SUBAPPLICATION Uebung_171c_ASR (* Exercise for ASR_AX_SR, ueber AE-Adapter mit logiBUS_IEA statt logiBUS_IE+AE_EVENT_TO_E *)
  (* Standard: 61499-2; Description: Copyright (c) 2026 Meisterschulen am Ostbahnhof This program and the accompanying materials are made available under the terms of the Eclipse Public License 2.0 which is available at https://www.eclipse.org/legal/epl-2.0/ SPDX-License-Identifier: EPL-2.0 *)
  (* Version 1.0, 2026-09-07, Franz Höpfinger, Meisterschulen am Ostbahnhof, initial API and implementation and/or initial documentation *)
  PACKAGE Uebungen;
  IMPORT logiBUS::io::DI::logiBUS_DI::Input_I1;
  IMPORT logiBUS::io::DI::logiBUS_DI::Input_I2;
  IMPORT logiBUS::io::DI::logiBUS_DI_Events::BUTTON_SINGLE_CLICK;
  IMPORT logiBUS::io::DQ::logiBUS_DO::Output_Q1;
  (* Documentation:
  SET/RESET über AE-Adapter mit logiBUS_IEA (AE bereits eingebaut)
   Dieselbe Funktion wie Uebung_171b_ASR, aber ohne die manuelle AE_EVENT_TO_E-Brücke pro Kanal: logiBUS_IEA ersetzt logiBUS_IE und liefert den AE-Plug (IN) bereits eingebaut - intern verdrahtet logiBUS_IEA genau das, was in 171b noch von Hand mit AE_EVENT_TO_E gebaut wurde.
   Funktionsbeschreibung
    - logiBUS_IEA kapselt intern einen logiBUS_IE und leitet dessen Klick-Events direkt auf einen eigenen AE-Plug (IN) um - derselbe Mechanismus wie IX → IXA für Pegelsignale, nur für Event-Eingänge.
   - ASR_2AE_TO_SR_1 bekommt seine SET_IN/RESET_IN jetzt direkt von den beiden logiBUS_IEA-Instanzen, ohne Zwischenbaustein.
    Arbeitsauftrag
   Testen Sie identisch zu Uebung_171_ASR/Uebung_171b_ASR: I1 klicken → Q1 EIN, I2 klicken → Q1 AUS. Vergleichen Sie alle drei SubApps im Editor: gleiches Verhalten, aber Uebung_171c_ASR kommt mit den wenigsten Bausteinen aus.
  *)
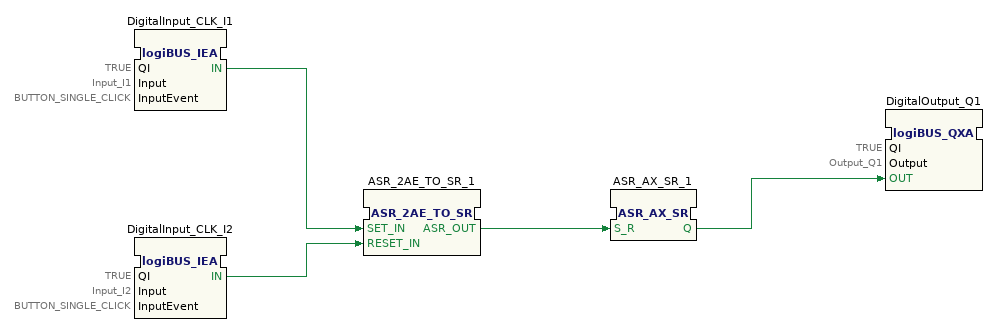
  (* Vergleich zu Uebung_171b_ASR: dort baute AE_EVENT_TO_E die Bruecke vom rohen logiBUS_IE-Klick-Event zum AE-Plug, manuell pro Kanal. Hier liefert logiBUS_IEA (statt logiBUS_IE) den AE-Plug bereits eingebaut - dieselbe Bruecke steckt schon im Baustein, kein separates AE_EVENT_TO_E noetig. *)
  FBS
    ASR_AX_SR_1 : adapter::events::unidirectional::ASR_AX_SR;
    ASR_2AE_TO_SR_1 : adapter::conversion::unidirectional::ASR_2AE_TO_SR;
    DigitalInput_CLK_I1 : logiBUS::io::DI::logiBUS_IEA(QI := TRUE, Input := Input_I1, InputEvent := BUTTON_SINGLE_CLICK);
    DigitalOutput_Q1 : logiBUS::io::DQ::logiBUS_QXA(QI := TRUE, Output := Output_Q1);
    DigitalInput_CLK_I2 : logiBUS::io::DI::logiBUS_IEA(QI := TRUE, Input := Input_I2, InputEvent := BUTTON_SINGLE_CLICK);
  END_FBS
  ADAPTER_CONNECTIONS
    DigitalInput_CLK_I1.IN TO ASR_2AE_TO_SR_1.SET_IN;
    DigitalInput_CLK_I2.IN TO ASR_2AE_TO_SR_1.RESET_IN;
    ASR_2AE_TO_SR_1.ASR_OUT TO ASR_AX_SR_1.S_R;
    ASR_AX_SR_1.Q TO DigitalOutput_Q1.OUT;
  END_CONNECTIONS
END_SUBAPPLICATION
